{attribute 'GeneratedUsingTerminal: EL3751-0000-0020'}
{attribute addProperty BoxType "EL3751-0000-0020"}
{attribute addProperty Id "StatusAT %I*Status_543010BE7"}
{attribute addProperty CRC "2924134660"}
{attribute addProperty Size "7"}
TYPE PAI_Status_Channel_AE4AC104 EXTENDS InputBase_8311D824 :
STRUCT
	{attribute addProperty Name "Status"}
	Status AT %I* : Status_543010BE;
END_STRUCT
END_TYPE

(* stored: Version 1.2.0.0, ProductVersion 3.1.4024.9
   DUT PAI_Status_Channel_AE4AC104: Id {b0b5fd06-9b7a-438a-bd2d-96f76a9836b2} *)
